PROGRAM MAIN
VAR
END_VAR

END_PROGRAM

(* stored: Version 1.1.0.1
   POU MAIN: Id {67756d31-ada2-403c-a4f9-99dee8df3d4e} *)
